# B&R Automation Studio project Laba4
Automation Studio 4.5.2.102; Default project; technology packages: Acp10Arnc0 5.2.1

## Configuration Real

### Task classes (Cpu.sw)
```
Cyclic#1 (cycle 2000 us, tolerance 0 us):
  ncsdcctrl <- ncsdcctrl.prg
  SDCAxisCtr <- SDCAxisCtrl_X.prg
  SDCAxisCt1 <- SDCAxisCtrl_Y.prg
  SDCAxisCt2 <- SDCAxisCtrl_Z.prg
Cyclic#4:
  User_Inter <- User_Interface.prg
DataObjects: Arnc0sys
NcDataObjects: AxisInit <- AxisInit.dob, gAxis03a <- gAxis03obj.gAxis03a.dob, gAxis03i <- gAxis03obj.gAxis03i.dob, AxisApt <- AxisApt.dob, gmcipvar <- GmcIpUserConfig.gmcipvar.dob, gmcipfun <- GmcIpUserConfig.gmcipfun.dob, gmcipfub <- GmcIpUserConfig.gmcipfub.dob, gmcipubr <- GmcIpUserConfig.gmcipubr.dob, gmcipusm <- GmcIpUserConfig.gmcipusm.dob, gmcipui <- GmcIpUserConfig.gmcipui.dob, gmcipus <- GmcIpUserConfig.gmcipus.dob, gmcipuc <- GmcIpUserConfig.gmcipuc.dob, gmcipsys <- GmcIpConfig.gmcipsys.dob, gmciplbr <- GmcIpConfig.gmciplbr.dob, gmcipcbr <- GmcIpConfig.gmcipcbr.dob, gmciplsm <- GmcIpConfig.gmciplsm.dob, gmcipcsm <- GmcIpConfig.gmcipcsm.dob, gmcipcfg <- GmcIpConfig.gmcipcfg.dob, gmcipiec <- GmcIpConfig.gmcipiec.dob, gmciplog <- GmcIpConfig.gmciplog.dob, gmcipesm <- GmcIpConfig.gmcipesm.dob, gmcipmxd <- GmcIpConfig.gmcipmxd.dob, gmcipmx <- GmcIpConfig.gmcipmx.dob, CncInit <- CncInit.dob, CncProg <- CncProg.dob, CncProg1 <- CncProg1.dob
VcDataObjects: Visu <- Visu.dob
Binaries: TCData, Acp10map1, acp10cfg, Acp10map, arconfig, User, Role, sysconf, iomap, asfw, ashwd, arnc0cfg, Arnc0map
Libraries: Acp10sdc, Library, Acp10man, Acp10_MC, sys_lib, brsystem, asstring, powerlnk, asieccon, AsMath, Arnc0man, DataObj, AsArLog, FileIO, AsArProf, AsMem, Runtime, astime, Acp10par, NcGlobal, asiotime, Acp10sim
```

### Hardware
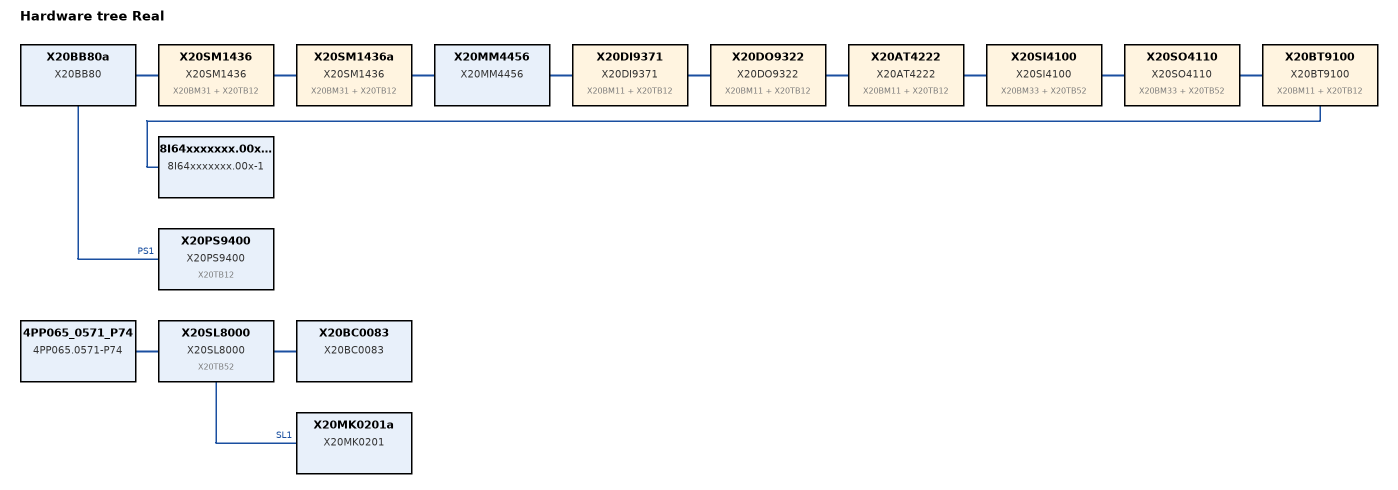
```
4PP065_0571_P74 : 4PP065.0571-P74 v1.1.2.0
  Connector IF4:
    Channel1
    ChannelID1 = McAcpBroadcast
    ChannelType1 = OCTET[96]
  Connector IF5:
    ActivateDevice = 1
    Mode = Manual
    InternetAddress = 10.0.1.10
    SubnetMask = 255.255.255.0
  ConfigurationID = labBR
  TimerDeviceType = EPLX2X
  TimerDevice = 4PP065_0571_P74.IF4
  TaskClassIdleTime = 2000
  Cyclic1Duration = 2000
  Cyclic1Tolerance = 0
  Cyclic1Output = 1
  Cyclic3Tolerance = 0
  VcObjectName = Visu
8I64xxxxxxx.00x-1 : 8I64xxxxxxx.00x-1 v1.3.9.1  [X2X1 -> X20BT9100.X2X1 [Cable Type=X2XCable, Length=10, Version=1.0.0.2]]
  BothEndSwitchesAreNormallyOpen_r1 = on
  QuickStopIsNormallyOpen_r1 = on
X20AT4222 : X20AT4222 v1.2.3.0  [SS1 -> X20TB12f.SS; SL -> X20BM11c.SL1]
X20BB80a : X20BB80 v1.0.2.0
X20BC0083 : X20BC0083 v2.7.0.0  [PLK1 -> X20SL8000.PLK2 (NodeNumber=2) [Cable Type=PowerlinkCable, Length=10, Version=1.0.0.2]; SL -> X20BB80a.SL1]
X20BM11a : X20BM11 v1.0.0.1  [X2X1 -> X20MM4456.X2X2]
X20BM11b : X20BM11 v1.0.0.1  [X2X1 -> X20BM11a.X2X2]
X20BM11c : X20BM11 v1.0.0.1  [X2X1 -> X20BM11b.X2X2]
X20BM11d : X20BM11 v1.0.0.1  [X2X1 -> X20BM33b.X2X2]
X20BM31a : X20BM31 v1.0.0.1  [X2X1 -> X20BB80a.IF1]
X20BM31b : X20BM31 v1.0.0.1  [X2X1 -> X20BM31a.X2X2]
X20BM33a : X20BM33 v1.0.0.4  [X2X1 -> X20BM11c.X2X2]
X20BM33b : X20BM33 v1.0.0.4  [X2X1 -> X20BM33a.X2X2]
X20BT9100 : X20BT9100 v1.0.3.0  [SS1 -> X20TB12g.SS; SL -> X20BM11d.SL1]
X20DI9371 : X20DI9371 v1.0.2.0  [SS1 -> X20TB12d.SS; SL -> X20BM11a.SL1]
X20DO9322 : X20DO9322 v1.0.3.0  [SS1 -> X20TB12e.SS; SL -> X20BM11b.SL1]
X20MK0201a : X20MK0201 v1.0.0.0  [SL -> X20SL8000.SL1]
X20MM4456 : X20MM4456 v1.1.5.0  [X2X1 -> X20BM31b.X2X2]
X20PS9400 : X20PS9400 v1.0.2.4  [SS1 -> X20TB12b.SS; PS -> X20BB80a.PS1]
X20SI4100 : X20SI4100 v1.10.1.1  [SS1 -> X20TB52b.SS; SL -> X20BM33a.SL1]
X20SL8000 : X20SL8000 v1.6.5.1  [PLK1 -> 4PP065_0571_P74.IF4 (NodeNumber=1) [Cable Type=PowerlinkCable, Length=10, Version=1.0.0.2]; PLK2 -> X20BC0083.PLK1 (NodeNumber=1) [Cable Type=PowerlinkCable, Length=10, Version=1.0.0.2]; SS1 -> X20TB52a.SS]
  SafeProject = SafeLOGIC-1
X20SM1436 : X20SM1436 v1.4.2.1  [SS1 -> X20TB12a.SS; SL -> X20BM31a.SL1]
X20SM1436a : X20SM1436 v1.4.2.1  [SS1 -> X20TB12c.SS; SL -> X20BM31b.SL1]
X20SO4110 : X20SO4110 v1.10.1.1  [SS1 -> X20TB52c.SS; SL -> X20BM33b.SL1]
  SafeLogicID = 2
  SafeModuleID = 3
X20TB12a : X20TB12 v1.0.0.0
X20TB12b : X20TB12 v1.0.0.0
X20TB12c : X20TB12 v1.0.0.0
X20TB12d : X20TB12 v1.0.0.0
X20TB12e : X20TB12 v1.0.0.0
X20TB12f : X20TB12 v1.0.0.0
X20TB12g : X20TB12 v1.0.0.0
X20TB52a : X20TB52 v1.0.0.1
X20TB52b : X20TB52 v1.0.0.1
X20TB52c : X20TB52 v1.0.0.1
```

## Logical view

### Global.var
```iecst
VAR
	Trajectory : FB_Trajectory := (0);
	Move_axis : FB_move := (0);
	Power_home : FB_power := (0);
	AxisX : ACP10AXIS_typ := (0);
	AxisX_EncIf : SdcEncIf16_typ := (0);
	AxisX_DrvIf : SdcDrvIf16_typ := (0);
	AxisX_DiDoIf : SdcDiDoIf_typ := (0);
	AxisX_HW : SdcHwCfg_typ := (0);
	AxisY : ACP10AXIS_typ := (0);
	AxisY_EncIf : SdcEncIf16_typ := (0);
	AxisY_DrvIf : SdcDrvIf16_typ := (0);
	AxisY_DiDoIf : SdcDiDoIf_typ := (0);
	AxisY_HW : SdcHwCfg_typ := (0);
	AxisZ : ACP10AXIS_typ := (0);
	AxisZ_EncIf : SdcEncIf16_typ := (0);
	AxisZ_DrvIf : SdcDrvIf16_typ := (0);
	AxisZ_DiDoIf : SdcDiDoIf_typ := (0);
	AxisZ_HW : SdcHwCfg_typ := (0);
	gAxis01 : ACP10AXIS_typ := (0);
	gAxis02 : ACP10AXIS_typ := (0);
	gAxisTest : ACP10AXIS_typ := (0);
	gAxisTest_HW : SdcHwCfg_typ := (0);
	gAxisTest_DrvIf : SdcDrvIf16_typ := (0);
	gAxisTest_DiDoIf : SdcDiDoIf_typ := (0);
	gAxisTest_ModuleOk : BOOL := 0;
	gAxis03 : ACP10AXIS_typ := (0);
	gAxis03_HW : SdcHwCfg_typ := (0);
	gAxis03_DrvIf : SdcDrvIf16_typ := (0);
	gAxis03_DiDoIf : SdcDiDoIf_typ := (0);
	gAxis03_ModuleOk : BOOL := 0;
	CNCsys : ARNC0CNC_typ;
END_VAR
```

### Program Logical/User_Interface

#### Variables.var
```iecst
VAR
	length : UINT := 0;
	homing : MC_Home := (0);
	power : MC_Power := (0);
END_VAR
```

#### Main.c
```c
#include <bur/plctypes.h>

#ifdef _DEFAULT_INCLUDES
	#include <AsDefault.h>
#endif

void _INIT ProgramInit(void)
{
	Trajectory.AxisY = &AxisY;
	Trajectory.AxisZ = &AxisZ;
	Trajectory.lengthY = 0;
	Trajectory.lengthZ = 0;
	Move_axis.length = 0;
}

void _CYCLIC ProgramCyclic(void)
{
	FB_Trajectory(&Trajectory);
}

void _EXIT ProgramExit(void)
{

}
```
